{attribute 'qualified_only'}
{attribute 'strict'}
{attribute 'to_string'}
TYPE E_Mode :
(
	manual,
	automatic
);
END_TYPE

(* stored: Version 1.1.0.1
   DUT E_Mode: Id {23ac1c79-175e-43cc-8a14-61266fdb4bfe} *)
